// This function has been automatically generated from the project information.
VAR_GLOBAL CONSTANT
	{attribute 'const_non_replaced'}
	stLibVersion_Base_PLC : ST_LibVersion := (iMajor := 0, iMinor := 3, iBuild := 5, iRevision := 6, sVersion := '0.3.5.6');
END_VAR

(* stored: Version 1.1.0.1, ProductVersion 3.1.0.26
   GVL Global_Version: Id {db682a82-4552-4aea-8efb-452bbfc07dbc} *)
